// TIA Portal project "hello-world" (V17)

(* hardware
DEVICE "S7-1500/ET200MP station_1"  S7-1500 station
   slot 0: "Rail_0"  Rack  6ES7 590-1***0-0AA0
   slot 1: "PLC_1"  CPU 1511-1 PN  6ES7 511-1AK02-0AB0  V2.9
      slot 3: "CPU display_1"  6ES7591-1AA00-0AA0
      slot 32768: "PROFINET interface_1"  X1
         slot 32769: "Port_1"  X1 P1
         slot 32770: "Port_2"  X1 P2
      slot 34817: "Virtual CP interface port_1"  Virtual CP interface port  Virtual CP interface port
*)

// ===== PLC "PLC_1"  CPU 1511-1 PN =====

DATA_BLOCK "Devices"   // DB1
{ S7_Optimized_Access := 'TRUE' }
VERSION : 0.1
   VAR
      MOTOR1 : Struct
         START : Bool;
         STOP : Bool;
         RUNNING : Bool;
         ERROR : Bool;
         OVERLOAD : Bool;
      END_STRUCT;
   END_VAR
BEGIN
END_DATA_BLOCK

ORGANIZATION_BLOCK "Main"   // OB1, LAD, ProgramCycle
TITLE = "Main Program Sweep (Cycle)"
{ S7_Optimized_Access := 'TRUE' }
VERSION : 0.1
   VAR_INPUT
      Initial_Call : Bool;   // Initial call of this OB
      Remanence : Bool;   // =True, if remanent data are available
   END_VAR
BEGIN

REGION Network 1: CONTROL MOTOR 1
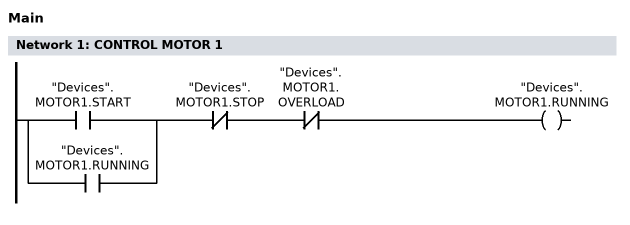
   RUNG wire#powerrail
      Contact( "Devices".MOTOR1.START )
      wire#w1
      I_Contact( "Devices".MOTOR1.STOP )
      I_Contact( "Devices".MOTOR1.OVERLOAD )
      Coil( "Devices".MOTOR1.RUNNING )
   END_RUNG
   RUNG wire#powerrail
      Contact( "Devices".MOTOR1.RUNNING )
   END_RUNG wire#w1
   // the same network as SCL:
   "Devices".MOTOR1.RUNNING := ("Devices".MOTOR1.START OR "Devices".MOTOR1.RUNNING) AND NOT "Devices".MOTOR1.STOP AND NOT "Devices".MOTOR1.OVERLOAD;
END_REGION
END_ORGANIZATION_BLOCK